Staubli VAL3: timerDialog.pgx

public program timerDialog(string x_sMsg, num x_nTime)
  local num l_nTime
  local num l_nStartLine
  local num l_nLine
  local num i
  local string l_sMessage
begin
  //
  // use for other task
  //
  if watch(bShowDialog==false,3)==false
    bShowDialog=false
    return
  else
    setMutex(bShowDialog)
    //
    //call listempty()
    //
    l_nTime=clock()
    call stringCopy(x_sMsg,sMessage)
    call divideString(sMessage,l_nLine)
    l_nStartLine=round(5-l_nLine/2)
    do
      // Start LINE
      call type(0,l_nStartLine-2,"┌──────────────────────────────────────┐")
      call type(0,l_nStartLine-1,"│                                      │")
      // write the message
      for i=0 to l_nLine
        call type(0,l_nStartLine+i,"")
        call type(39,l_nStartLine+i,"")
        //call typeCenter(i+l_nStartLine,sMessage[i],38,false)
        l_sMessage=sMessage[i]
        call typeCenter(i+l_nStartLine,l_sMessage,38,false)
        call type(0,l_nStartLine+i,"│"+l_sMessage+"│")
      endFor
      // end LINE
      call type(0,l_nStartLine+l_nLine+1,"│                                      │")
      call type(0,l_nStartLine+l_nLine+2,"└──────────────────────────────────────┘")
      // release
      if x_nTime==0
        delay(0.1)
      else
        delay(0)
      endIf
    until (clock()-l_nTime)>=x_nTime
    //
    bShowDialog=false
    bUseRefresh=true
  endIf
end
